// TwinCAT 3 PLC project MainPlc
// ProgramVersion: 3.1.4023.0
// libraries:
//   Tc2_Standard, * (Beckhoff Automation GmbH)
//   Tc2_System, * (Beckhoff Automation GmbH)
//   Tc3_Module, * (Beckhoff Automation GmbH)
// project tree:
//   App/Components/ fbPneumaticActuator.TcPOU, stComponents.TcDUT
//   App/Data/ fcEvalConitinuos.TcPOU, stContinuosValueData.TcDUT (not stored), stData.TcDUT (not stored)
//   App/ enumMode.TcDUT, fbStation.TcPOU, MAIN.TcPOU
//   / PlcTask.TcTTO

CONFIGURATION MainPlc
    RESOURCE PLC ON TwinCAT3
        TASK PlcTask(INTERVAL := T#10ms, PRIORITY := 20);
        PROGRAM MAIN WITH PlcTask : MAIN;
    END_RESOURCE
END_CONFIGURATION

// ---- App/Components/stComponents.TcDUT
{attribute wpf [Container(Layout.Stack)]}
{attribute addProperty Name "<#Components#>"}
TYPE stComponents :
STRUCT	
	{attribute addProperty Name "<#Horizontal piston#> A1"}	
	_horizontalPiston : fbPneumaticActuator;
	{attribute addProperty Name "<#Vertical piston#> A2"}
	_verticalPiston : fbPneumaticActuator;
	{attribute addProperty Name "<#Gripper#> A3"}
	_gripper : fbPneumaticActuator;
	{attribute addProperty Name "<#Locker#> A4"}
	_horizontalPistonLockerFailed : fbPneumaticActuator;
END_STRUCT
END_TYPE

// ---- App/enumMode.TcDUT
{attribute 'qualified_only'}
{attribute 'strict'}
TYPE enumMode :
(
	None := 0,
	Ground := 10,
	Automat := 20,
	Manual := 30
);
END_TYPE

// ---- App/MAIN.TcPOU
PROGRAM MAIN
VAR
	_station : fbStation;	
END_VAR

_station();

END_PROGRAM

// ---- App/fbStation.TcPOU
{attribute wpf [Container(Layout.Tabs)]}
FUNCTION_BLOCK fbStation
VAR		
	{attribute wpf [Container(Layout.Stack)]}
	{attribute addProperty Name "<#Select mode#>"}
	_modeSelector : enumMode;
	{attribute clr [ReadOnly()]}
	{attribute addProperty Name "<#CurrentMode#>"}
	_modeCurrent : enumMode;
		
	{attribute addProperty Name "<#Step description#>"}
	_stepInfo : STRING[255];
	
	{attribute addProperty Name "<#Error description#>"}
	_errorInfo : STRING[255];
	
	{attribute addProperty Name "<#Components#>"}
	_components : stComponents;
	
	{attribute addProperty Name "<#Data#>"}
	_data : stData;
END_VAR


_errorInfo := '<#No Error#>';

_modeCurrent := _modeSelector;

CASE _modeCurrent OF
	enumMode.Ground :
		GroundMode();
	enumMode.Automat :
		AutomatMode();
	enumMode.Manual:
		ManualMode();	
END_CASE

METHOD AutomatMode

VAR_INST
	_step : INT;
	_isOk : BOOL;	
END_VAR
CASE _step OF
	0:		
		_stepInfo := '<#Checking base position#>';		
		IF(_components._verticalPiston.Retract() 
		AND_THEN _components._gripper.Extend() 
		AND_THEN _components._horizontalPiston.Retract()) 
		THEN
			_step := 100;		
		END_IF
	100:
	   _stepInfo := '<#Measure the parameters.#>';
	   _isOk := fcEvalConitinuos(Val := 0.0, Data := _data.DimX)
				AND fcEvalConitinuos(Val := 0.0, Data := _data.DimY)
				AND fcEvalConitinuos(Val := 0.0, Data := _data.DimZ);

		_step := 200;				
	200:
		_stepInfo := '<#Take entity#>';
		IF(_components._verticalPiston.Extend() 
		AND_THEN _components._gripper.Retract())
		THEN
			IF _isOK THEN
				_step := 300;
			ELSE	
				_step := 500;
			END_IF;	
		END_IF;   
	300:
		_stepInfo := '<#Move entity to Passed conveyor#>';
		IF(_components._horizontalPiston.Extend()
		AND_THEN _components._verticalPiston.Extend() 
		AND_THEN _components._gripper.Retract())
		THEN
			_step := 500;
		END_IF;		
	400:
		_stepInfo := '<#Move entity to Failed conveyor#>';
		IF(_components._horizontalPistonLockerFailed.Extend()
		AND_THEN _components._horizontalPiston.Extend()
		AND_THEN _components._verticalPiston.Extend() 
		AND_THEN _components._gripper.Retract())
		THEN
			_step := 500;
		END_IF;			
	500:
		_step := 0;	
END_CASE
END_METHOD

METHOD GroundMode : BOOL
VAR_INST
	_step : INT;
END_VAR
CASE _step OF
	0:		
		_stepInfo := '<#Moving everything to ground position#>';		
		IF(_components._verticalPiston.Retract() 
		AND_THEN _components._gripper.Extend() 
		AND_THEN _components._horizontalPiston.Retract()) 
		THEN
			_step := 100;		
		END_IF
	100:
	   _stepInfo := '<#All in position ready to start#>';
END_CASE
END_METHOD

METHOD ManualMode : BOOL
VAR_INPUT
END_VAR
_components._gripper.Manual();
_components._horizontalPiston.Manual();
_components._verticalPiston.Manual();
END_METHOD

END_FUNCTION_BLOCK

// ---- App/Data/fcEvalConitinuos.TcPOU
FUNCTION fcEvalConitinuos : BOOL
VAR_INPUT
	Val : REAL;
	Data : stContinuosValueData;
END_VAR
VAR
END_VAR

Data.Measured := Val;
fcEvalConitinuos := (Data.Mininum >= Data.Measured AND Data.Maximum <= Data.Measured);

END_FUNCTION

// ---- App/Components/fbPneumaticActuator.TcPOU
{attribute wpf [Container(Layout.Wrap)]}
{attribute wpf [Group(Layout.GroupBox)]}
FUNCTION_BLOCK fbPneumaticActuator
VAR_INPUT
	{attribute wpf [Container(Layout.Stack)]}	
	{attribute addProperty Name "Retracted"}
	{attribute addProperty ToolTip "Sensor indicating that the actuator is retracted"}
	inRetracted : BOOL;	
	{attribute addProperty Name "Extend"}
	{attribute addProperty ToolTip "Sensor indicating that the actuator is extended"}
	inExtended : BOOL;	
END_VAR
VAR_OUTPUT
	{attribute wpf [Container(Layout.Stack)]}
	{attribute addProperty Name "Retract"}
	{attribute addProperty ToolTip "Signal for retracting"}
	outRetract : BOOL;
	{attribute addProperty Name "Extend"}
	{attribute addProperty ToolTip "Signal for Extending"}
	outExtend : BOOL;
END_VAR
VAR
	{attribute wpf [Container(Layout.UniformGrid)]}
	{attribute addProperty Name "Manual Retract"}
	{attribute addProperty ToolTip "Executes retraction in manual mode"}
	_manualRetract : BOOL;
	{attribute addProperty Name "Manual Extend"}
	{attribute addProperty ToolTip "Executes extension in manual mode"}
	_manualExtend : BOOL;
END_VAR

METHOD Extend : BOOL
THIS^.outRetract := FALSE;
THIS^.outExtend := TRUE;

Extend := THIS^.inExtended;
END_METHOD

METHOD Manual
IF(THIS^._manualExtend AND_THEN THIS^.Extend()) THEN THIS^._manualExtend := FALSE; END_IF;
IF(THIS^._manualRetract AND_THEN THIS^.Retract()) THEN THIS^._manualRetract := FALSE; END_IF;
END_METHOD

METHOD Retract : BOOL
THIS^.outRetract := TRUE;
THIS^.outExtend := FALSE;

Retract := THIS^.inRetracted;
END_METHOD

END_FUNCTION_BLOCK
